Universal Robots URScript: all_bows.script

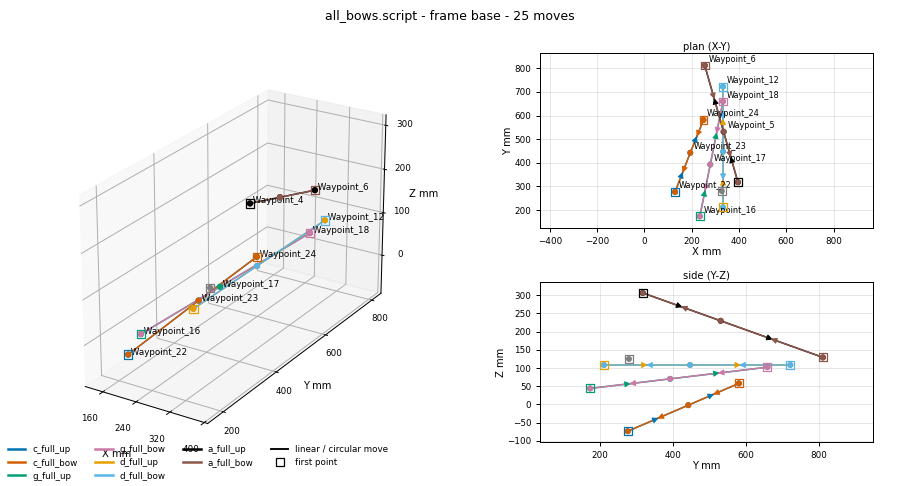
[picture p0: tool path of all_bows.script in frame base, 25 of 25 moves have a stored position in this frame; points joined in program order, loops and branches not executed]
def unnamed():
  global _hidden_verificationVariable=0
  step_count_a36665b5_09a7_4590_bfbd_dbd8a2b6012c = 0.0
  thread Step_Counter_Thread_cd0368b8_8cd3_4a3c_9e82_82e3b543d6f5():
    while (True):
      step_count_a36665b5_09a7_4590_bfbd_dbd8a2b6012c = step_count_a36665b5_09a7_4590_bfbd_dbd8a2b6012c + 1.0
      sync()
    end
  end
  run Step_Counter_Thread_cd0368b8_8cd3_4a3c_9e82_82e3b543d6f5()
  set_standard_analog_input_domain(0, 1)
  set_standard_analog_input_domain(1, 1)
  set_tool_analog_input_domain(0, 1)
  set_tool_analog_input_domain(1, 1)
  set_analog_outputdomain(0, 0)
  set_analog_outputdomain(1, 0)
  set_input_actions_to_default()
  set_safety_mode_transition_hardness(1)
  set_target_payload(0.260000, [0.050000, -0.008000, 0.024000], [0.000163, 0.000163, 0.000163, 0.000000, 0.000000, 0.000000])
  set_gravity([0.0, 0.0, 9.82])
  set_tcp(p[0.028210348281514253,-0.09610723587300697,-0.09969041498611403,0.0,0.0,0.0])
  set_tool_communication(False, 115200, 0, 1, 1.5, 3.5)
  set_tool_output_mode(0)
  set_tool_digital_output_mode(0, 1)
  set_tool_digital_output_mode(1, 1)
  set_tool_voltage(0)
  global Plane_1=p[0.32571614183608727,0.7933870146316717,0.11820742021636722,-2.208244884171713,-0.24738609815952348,-1.9195085473101943]
  global Plane_2=p[0.3436052139151623,0.7478032414335104,0.10077839665899768,2.768545736097797,0.1284831553507919,1.3672805628273381]
  global Plane_3=p[0.31945151854627996,0.6757990361168175,0.09459088830114093,2.7301760593116526,-0.049483824131046385,1.4252239353300047]
  global Plane_4=p[0.3372257363094211,0.6222230974198586,0.07001667903587716,2.621672423508307,-0.12240385890263918,1.4373011913128484]
  # begin: URCap Installation Node
  #   Source: External Control, 1.0.5, FZI Research Center for Information Technology
  #   Type: External Control
  # end: URCap Installation Node
  global Waypoint_25_p=p[.327441175739, .280063197287, .124800697874, -1.835968163317, -1.627478693982, .236736499086]
  global Waypoint_25_q=[-2.863450715987023, -0.8779325517585104, 2.2021820451163023, -2.390852458908271, -1.0567741990394062, -2.8730427834273335]
  global Waypoint_22_p=p[.129484250144, .276804006919, -.073202509131, -1.835637292008, -1.631750632514, .239885997621]
  global Waypoint_22_q=[-2.680851761494772, -0.15272171915087895, 2.31638747850527, -3.331407209435934, -0.9844964186297815, -2.6800459066974085]
  global Waypoint_23_p=p[.193788862268, .442604658512, -.001862808906, -1.842389053539, -1.496635858153, .142094638695]
  global Waypoint_23_q=[-2.412469880534173, -0.4082673028383157, 2.0249265615986904, -3.095022597467647, -0.8032725526097568, -2.2372652714417924]
  global Waypoint_24_p=p[.249582907829, .581405619494, .057868196739, -1.842365216747, -1.383032382737, .062670771415]
  global Waypoint_24_q=[-2.301014021200069, -0.4292136371382069, 1.6474302572409938, -2.9438729370209384, -0.74218409639127, -1.9442029158929852]
  global Waypoint_19_p=p[.249582907829, .581405619494, .057868196739, -1.842365216747, -1.383032382737, .062670771415]
  global Waypoint_19_q=[-2.301014021200069, -0.4292136371382069, 1.6474302572409938, -2.9438729370209384, -0.74218409639127, -1.9442029158929852]
  global Waypoint_20_p=p[.193788862268, .442604658512, -.001862808906, -1.842389053539, -1.496635858153, .142094638695]
  global Waypoint_20_q=[-2.412469880534173, -0.4082673028383157, 2.0249265615986904, -3.095022597467647, -0.8032725526097568, -2.2372652714417924]
  global Waypoint_21_p=p[.129484250144, .276804006919, -.073202509131, -1.835637292008, -1.631750632514, .239885997621]
  global Waypoint_21_q=[-2.680851761494772, -0.15272171915087895, 2.31638747850527, -3.331407209435934, -0.9844964186297815, -2.6800459066974085]
  global Waypoint_16_p=p[.234239698429, .173482767533, .044020522270, -1.748553022590, -1.966156862980, .873741563229]
  global Waypoint_16_q=[-3.0913494447061822, -0.6894588925344856, 2.476797028131698, -2.636710781839504, -1.740481970217937, -3.1375743380598466]
  global Waypoint_17_p=p[.278373130956, .392903749619, .070316048888, -1.730968296797, -1.856181704588, .761951257439]
  global Waypoint_17_q=[-2.5968696306336376, -0.7386435216100811, 2.0489904531773684, -2.173591572816089, -1.2680291843104552, -2.7737850347270525]
  global Waypoint_18_p=p[.332008886777, .659568034338, .102273237896, -1.702060684636, -1.721742670087, .631106118068]
  global Waypoint_18_q=[-2.3092736795250994, -0.48309022847596506, 1.270759508735778, -1.8161087745438396, -0.9292687732931482, -2.5009753359650193]
  global Waypoint_13_p=p[.332008886777, .659568034338, .102273237896, -1.702060684636, -1.721742670087, .631106118068]
  global Waypoint_13_q=[-2.3092736795250994, -0.48309022847596506, 1.270759508735778, -1.8161087745438396, -0.9292687732931482, -2.5009753359650193]
  global Waypoint_14_p=p[.278373130956, .392903749619, .070316048888, -1.730968296797, -1.856181704588, .761951257439]
  global Waypoint_14_q=[-2.5968696306336376, -0.7386435216100811, 2.0489904531773684, -2.173591572816089, -1.2680291843104552, -2.7737850347270525]
  global Waypoint_15_p=p[.234239698429, .173482767533, .044020522270, -1.748553022590, -1.966156862980, .873741563229]
  global Waypoint_15_q=[-3.0913494447061822, -0.6894588925344856, 2.476797028131698, -2.636710781839504, -1.740481970217937, -3.1375743380598466]
  global Waypoint_10_p=p[.332580873770, .211379769050, .108291185252, -1.644956384976, -2.108101752358, 1.059071402912]
  global Waypoint_10_q=[-2.999210159655675, -0.9044912918890518, 2.2177420085479818, -2.1298181728944527, -1.8609334123373777, -3.1238684621592654]
  global Waypoint_11_p=p[.332299124832, .447473035233, .108291185236, -1.644956384993, -2.108101752396, 1.059071402850]
  global Waypoint_11_q=[-2.560621659761836, -0.762511368631869, 1.7887822200831496, -1.7990925777647124, -1.5512054499803334, -2.810039268405372]
  global Waypoint_12_p=p[.331971133677, .722315253805, .108291185217, -1.644956385012, -2.108101752441, 1.059071402778]
  global Waypoint_12_q=[-2.2638438383685493, -0.37471242368733115, 0.9072483221637506, -1.3311255735210121, -1.3414958159076118, -2.600104633961808]
  global Waypoint_7_p=p[.331971133677, .722315253805, .108291185217, -1.644956385012, -2.108101752441, 1.059071402778]
  global Waypoint_7_q=[-2.2638438383685493, -0.37471242368733115, 0.9072483221637506, -1.3311255735210121, -1.3414958159076118, -2.600104633961808]
  global Waypoint_8_p=p[.332299124832, .447473035233, .108291185236, -1.644956384993, -2.108101752396, 1.059071402850]
  global Waypoint_8_q=[-2.560621659761836, -0.762511368631869, 1.7887822200831496, -1.7990925777647124, -1.5512054499803334, -2.810039268405372]
  global Waypoint_9_p=p[.332580873770, .211379769050, .108291185252, -1.644956384976, -2.108101752358, 1.059071402912]
  global Waypoint_9_q=[-2.999210159655675, -0.9044912918890518, 2.2177420085479818, -2.1298181728944527, -1.8609334123373777, -3.1238684621592654]
  global Waypoint_4_p=p[.395327225653, .317909637846, .305826489206, 1.738924283763, 2.310428550894, -1.107753568900]
  global Waypoint_4_q=[-2.8159710998724172, -1.1839948226902983, 1.8074412843478633, -1.5759268018043278, -1.9904723215831952, -2.957970419382864]
  global Waypoint_5_p=p[.334760756351, .531331188399, .229440537136, 1.738924283776, 2.310428550993, -1.107753568706]
  global Waypoint_5_q=[-2.4598168785017207, -0.8870623512050804, 1.5263397184716765, -1.4998985637660107, -1.7695796214075479, -2.663439034730976]
  global Waypoint_6_p=p[.255207331122, .811658167337, .129108386415, 1.738924283794, 2.310428551122, -1.107753568452]
  global Waypoint_6_q=[-2.1357390865281953, -0.25800854558481134, 0.5461371958945197, -1.125392426618962, -1.555786650509841, -2.419880619474636]
  global Waypoint_1_p=p[.255207331122, .811658167337, .129108386415, 1.738924283794, 2.310428551122, -1.107753568452]
  global Waypoint_1_q=[-2.1357390865281953, -0.25800854558481134, 0.5461371958945197, -1.125392426618962, -1.555786650509841, -2.419880619474636]
  global Waypoint_3_p=p[.334760756351, .531331188399, .229440537136, 1.738924283776, 2.310428550993, -1.107753568706]
  global Waypoint_3_q=[-2.4598168785017207, -0.8870623512050804, 1.5263397184716765, -1.4998985637660107, -1.7695796214075479, -2.663439034730976]
  global Waypoint_2_p=p[.395327225653, .317909637846, .305826489206, 1.738924283763, 2.310428550894, -1.107753568900]
  global Waypoint_2_q=[-2.8159710998724172, -1.1839948226902983, 1.8074412843478633, -1.5759268018043278, -1.9904723215831952, -2.957970419382864]
  def c_full_up():
    $ 13 "c_full_up" "noBreak"
    $ 14 "MoveL"
    $ 15 "Waypoint_22" "breakAfter"
    movel(Waypoint_22_p, a=1.2, v=0.25)
    $ 16 "Waypoint_23" "breakAfter"
    movel(Waypoint_23_p, a=1.2, v=0.25, r=0.05)
    $ 17 "Waypoint_24" "breakAfter"
    movel(Waypoint_24_p, a=1.2, v=0.25)
  end
  def c_full_bow():
    $ 18 "c_full_bow" "noBreak"
    $ 19 "MoveL"
    $ 20 "Waypoint_19" "breakAfter"
    movel(Waypoint_19_p, a=1.2, v=0.25)
    $ 21 "Waypoint_20" "breakAfter"
    movel(Waypoint_20_p, a=1.2, v=0.25, r=0.05)
    $ 22 "Waypoint_21" "breakAfter"
    movel(Waypoint_21_p, a=1.2, v=0.25)
  end
  def g_full_up():
    $ 23 "g_full_up" "noBreak"
    $ 24 "MoveL"
    $ 25 "Waypoint_16" "breakAfter"
    movel(Waypoint_16_p, a=1.2, v=0.25)
    $ 26 "Waypoint_17" "breakAfter"
    movel(Waypoint_17_p, a=1.2, v=0.25, r=0.05)
    $ 27 "Waypoint_18" "breakAfter"
    movel(Waypoint_18_p, a=1.2, v=0.25)
  end
  def g_full_bow():
    $ 28 "g_full_bow" "noBreak"
    $ 29 "MoveL"
    $ 30 "Waypoint_13" "breakAfter"
    movel(Waypoint_13_p, a=1.2, v=0.25)
    $ 31 "Waypoint_14" "breakAfter"
    movel(Waypoint_14_p, a=1.2, v=0.25, r=0.05)
    $ 32 "Waypoint_15" "breakAfter"
    movel(Waypoint_15_p, a=1.2, v=0.25)
  end
  def d_full_up():
    $ 33 "d_full_up" "noBreak"
    $ 34 "MoveL"
    $ 35 "Waypoint_10" "breakAfter"
    movel(Waypoint_10_p, a=1.2, v=0.25)
    $ 36 "Waypoint_11" "breakAfter"
    movel(Waypoint_11_p, a=1.2, v=0.25, r=0.05)
    $ 37 "Waypoint_12" "breakAfter"
    movel(Waypoint_12_p, a=1.2, v=0.25)
  end
  def d_full_bow():
    $ 38 "d_full_bow" "noBreak"
    $ 39 "MoveL"
    $ 40 "Waypoint_7" "breakAfter"
    movel(Waypoint_7_p, a=1.2, v=0.25)
    $ 41 "Waypoint_8" "breakAfter"
    movel(Waypoint_8_p, a=1.2, v=0.25, r=0.05)
    $ 42 "Waypoint_9" "breakAfter"
    movel(Waypoint_9_p, a=1.2, v=0.25)
  end
  def a_full_up():
    $ 43 "a_full_up" "noBreak"
    $ 44 "MoveL"
    $ 45 "Waypoint_4" "breakAfter"
    movel(Waypoint_4_p, a=1.2, v=0.25)
    $ 46 "Waypoint_5" "breakAfter"
    movel(Waypoint_5_p, a=1.2, v=0.25, r=0.05)
    $ 47 "Waypoint_6" "breakAfter"
    movel(Waypoint_6_p, a=1.2, v=0.25)
  end
  def a_full_bow():
    $ 48 "a_full_bow" "noBreak"
    $ 49 "MoveL"
    $ 50 "Waypoint_1" "breakAfter"
    movel(Waypoint_1_p, a=1.2, v=0.25)
    $ 51 "Waypoint_3" "breakAfter"
    movel(Waypoint_3_p, a=1.2, v=0.25, r=0.05)
    $ 52 "Waypoint_2" "breakAfter"
    movel(Waypoint_2_p, a=1.2, v=0.25)
  end
  while (True):
    $ 2 "Robot Program"
    $ 3 "MoveJ"
    $ 4 "Waypoint_25" "breakAfter"
    movej(get_inverse_kin(Waypoint_25_p, qnear=Waypoint_25_q), a=1.3962634015954636, v=1.0471975511965976)
    $ 5 "Call a_full_bow"
    a_full_bow()
    $ 6 "Call a_full_up"
    a_full_up()
    $ 7 "Call d_full_bow"
    d_full_bow()
    $ 8 "Call d_full_up"
    d_full_up()
    $ 9 "Call g_full_bow"
    g_full_bow()
    $ 10 "Call g_full_up"
    g_full_up()
    $ 11 "Call c_full_bow"
    c_full_bow()
    $ 12 "Call c_full_up"
    c_full_up()
  end
end
